(* IEC 61131-3 sources: st2cc/examples, 4 files *)

(* ---- example.st ---- *)
PROGRAM Main
    VAR
        sensor0 AT %IX0.0: BOOL;
        sensor1 AT %IX0.1: BOOL;
        sensor2 AT %IX0.2: BOOL;
        actuator0 AT %QX0.0: BOOL;
        actuator1 AT %QX0.1: BOOL;
    END_VAR
    IF sensor0 OR (sensor1 AND sensor2) THEN
        actuator0 := TRUE;
        actuator1 := TRUE;
    ELSE
        actuator0 := FALSE;
        actuator1 := FALSE;
    END_IF
END_PROGRAM

(* ---- example2.st ---- *)
PROGRAM Main
    VAR
        start_button: BOOL;
        motor_on: BOOL;
        temp_sensor: INT;
        valve_ctrl: INT;
    END_VAR
    IF start_button THEN
        motor_on := TRUE;
    ELSE
        motor_on := FALSE;
    END_IF
    valve_ctrl := temp_sensor * 2;
END_PROGRAM

// TODO
// StartButton AT %I0.0: BOOL;
// MotorOn AT %Q0.0: BOOL;
// TempSensor AT %IW2: REAL;
// ValveCtrl AT %QW4: REAL;

(* ---- record.st ---- *)
TYPE
    Point: STRUCT
        x: REAL;
        y: REAL;
    END_STRUCT;
END_TYPE

PROGRAM Main
    VAR
        p1: Point;
        p2: Point;
        distance: REAL;
    END_VAR

    p1.x := 3.0;
    p1.y := 4.0;

    p2.x := 6.0;
    p2.y := 8.0;

    distance := SQRT(POW(p2.x - p1.x, 2) + POW(p2.y - p1.y, 2));

END_PROGRAM

(* ---- recursion.st ---- *)
PROGRAM Main
    VAR
        n AT %IW0: INT;
        result AT %QW0: INT;
    END_VAR
    result := Factorial(n);
END_PROGRAM

FUNCTION Factorial: INT
    VAR_INPUT
        num: INT;
    END_VAR
    IF num <= 1 THEN
        Factorial := 1;
    ELSE
        Factorial := num * Factorial(num - 1);
    END_IF
END_FUNCTION
